(* CODESYS project SemaforoSimples.project

Project tree, tasks and I/O mapping:
  Device : CODESYS Control Win V3 x64, 3S - Smart Software Solutions GmbH, version 3.5.11.30
    application Application
      libraries: Standard, * (System); Util, * (System)
      task MainTask (cyclic, interval t#20ms, priority 1) calls PLC_PRG
      task VISU_TASK (cyclic, interval 100 ms, priority 31) calls VisuElems.Visu_Prg
      program PLC_PRG [LD]
      visualisation Visualization
  libraries: VisuSymbols, 3.5.10.0 (System)
  text list GlobalTextList
*)

// Device/Application/PLC_PRG
PROGRAM PLC_PRG
VAR
	// INPUTS
	startButton	: BOOL;
	stopButton	: BOOL;
	
	// OUTPUTS
	redLight	: BOOL;
	greenLight	: BOOL;
	yellowLight	: BOOL;
	
	onOff: SR;
	Enable: BOOL;

	timerRed: TON;
	timerGreen: TON;
	timerYellow: TON;
	blinkYellow: BLINK;
END_VAR

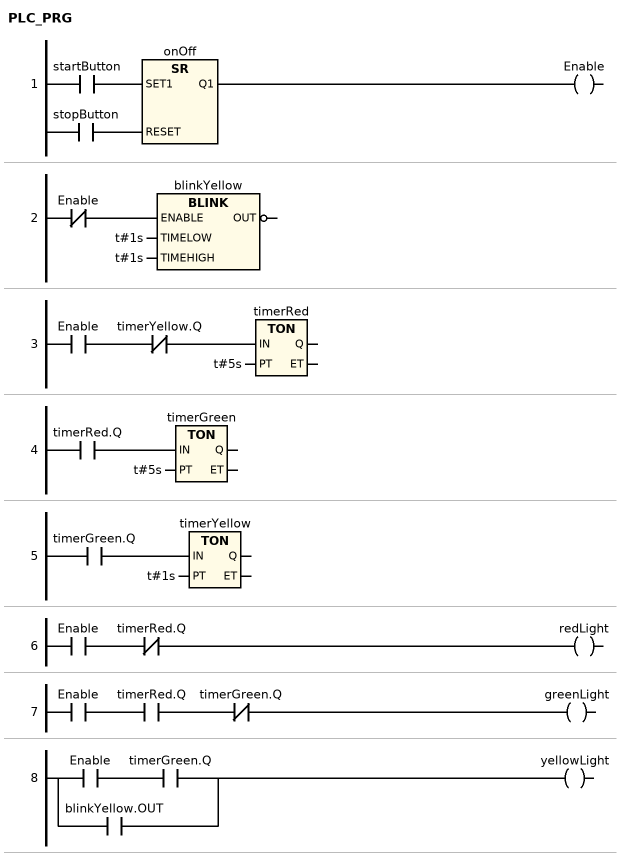
// NETWORK 1
onOff(SET1 := startButton, RESET := stopButton); // SR
Enable := onOff.Q1;

// NETWORK 2
blinkYellow(ENABLE := NOT Enable, TIMELOW := t#1s, TIMEHIGH := t#1s); // BLINK

// NETWORK 3
timerRed(IN := Enable AND NOT timerYellow.Q, PT := t#5s); // TON

// NETWORK 4
timerGreen(IN := timerRed.Q, PT := t#5s); // TON

// NETWORK 5
timerYellow(IN := timerGreen.Q, PT := t#1s); // TON

// NETWORK 6
redLight := Enable AND NOT timerRed.Q;

// NETWORK 7
greenLight := Enable AND timerRed.Q AND NOT timerGreen.Q;

// NETWORK 8
yellowLight := Enable AND timerGreen.Q OR blinkYellow.OUT;

END_PROGRAM

// Device/Application/Visualization
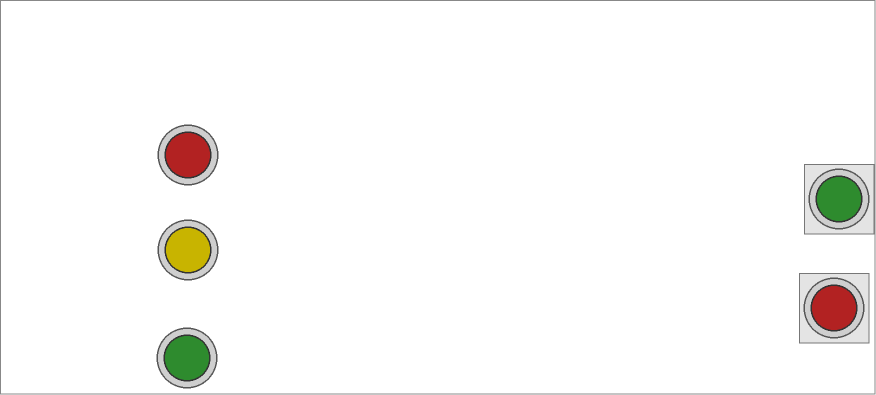
VISUALIZATION Visualization  // 876x395
    Lamp1 (153,120 70x70), variable: PLC_PRG.redLight, style: Lamp-Lamp1-Red
    Lamp1 (153,215 70x70), variable: PLC_PRG.yellowLight, style: Lamp-Lamp1-Yellow
    Lamp1 (152,323 70x70), variable: PLC_PRG.greenLight, style: Lamp-Lamp1-Green
    PushSwitch (804,164 70x70), variable: PLC_PRG.startButton, behaviour: TAP, style: Switch-PushSwitch-Green
    PushSwitch (799,273 70x70), variable: PLC_PRG.stopButton, behaviour: TAP, style: Switch-PushSwitch-Red
END_VISUALIZATION
